(* Logix 5000 project; controller _2081 vendor 1 type 14 code 77 rev 19.11; software revision 19.01 *)

TASK Continuous (continuous, watchdog 500 ms) : BGK_OVEN

MODULES
   Controller : vendor 1 type 14 code 77 (CompactLogixL32EController 0, rev 19.11)
      LocalENB : 1769-L32E Ethernet Port (CompactLogixL32Ethernet 1, rev 19.11)
      Local : CompactBus (CompactVirtualAdapter 3, rev 19.11)
         DC_Input_Slot_3 : 1769-IQ16 (Compact 3, rev 1.1, Input RPI 2 ms)
         DC_Input_Slot_4 : 1769-IQ16 (Compact 4, rev 1.1, Input RPI 2 ms)
         Relay_Out_Slot_5 : 1769-OW8I (Compact 5, rev 2.1, Output RPI 2 ms)
         Analog_Input : 1769-IF8 (Compact 1, rev 1.1, Output RPI 2 ms)
         Analog_Out : vendor 1 type 10 code 39 (Compact 2, rev 1.3, Output RPI 2 ms)
         Relay_Out_Slot_6 : 1769-OW8I (Compact 6, rev 2.1, Output RPI 2 ms)
END_MODULES

TYPE Conveyor :
STRUCT
   Conveyors_Input : PowerFlex_40_Status;
   Conveyor_Output : PowerFlex_40_Command;
END_STRUCT
END_TYPE

TYPE DeviceNETPowerFlex40 :
STRUCT
   Command : PowerFlex_40_Command;   // Start/Stop/Speed Etc.
   Status : PowerFlex_40_Status;   // Fault/Inputs Etc.
END_STRUCT
END_TYPE

TYPE PowerFlex_40_Command :
STRUCT
   Stop : BOOL;   // Stop=1
   Start : BOOL;   // Start=1
   Jog : BOOL;   // Jog=1
   Clear_Faults : BOOL;
   Direction_Forward : BOOL;
   Direction_Reverse : BOOL;
   Not_Used : BOOL;
   MOP_Increment : BOOL;
   Accel_Rate1 : BOOL;
   Accel_Rate2 : BOOL;
   Decel_Rate1 : BOOL;
   Decel_Rate2 : BOOL;
   Reference_Sel1 : BOOL;
   Reference_Sel2 : BOOL;
   Reference_Sel3 : BOOL;
   MOP_Decrement : BOOL;
   Speed_Command : INT;
END_STRUCT
END_TYPE

TYPE PowerFlex_40_Status :
STRUCT
   Ready : BOOL;   // Ready=1
   Active : BOOL;   // Active=1
   Command_Direction : BOOL;   // Forward=1
   Actual_Direction : BOOL;
   Accelerating : BOOL;
   Decelerating : BOOL;
   Alarm_Present : BOOL;
   Fault_Present : BOOL;
   At_Speed : BOOL;
   Main_Freq : BOOL;   // Comm Control=1
   Operation_Command : BOOL;   // Comm Control=1
   Parameters : BOOL;   // Locked=1
   Dig_In_1_Status : BOOL;   // Status of Input 1
   Dig_In_2_Status : BOOL;   // Status of Input 2
   Dig_In_3_Status : BOOL;   // Status of Input 3
   Dig_In_4_Status : BOOL;   // Status of Input 4
   Conveyor_Speed : INT;
END_STRUCT
END_TYPE

VAR_GLOBAL   (* controller tags *)
   Exhaust_Temp_PID : PID := (CTL := -2147446144, EN := 1, INI := 1, OLH := 1, DVPA := 1, PVHA := 1, SP := 300.0, KP := 15.0, KI := 0.2, MAXS := 932.0, MINS := 32.0, SO := 100.0, MAXO := 100.0, UPD := 0.5, PV := 297.0, ERR := 3.0, OUT := 100.0, MAXI := 932.0, MINI := 32.0, MAXCV := 300.0, MAXTIE := 4095.0, DATA[0] := 94.97618, DATA[1] := -471.1111, DATA[2] := 297.0, DATA[3] := 3.0, DATA[4] := 300.0, DATA[5] := 0.11111111, DATA[6] := 1.0, DATA[7] := 8.0, DATA[8] := 15.0, DATA[9] := 0.2, DATA[11] := 15.0, DATA[12] := 0.2, DATA[15] := 3.0, DATA[16] := 0.024420025);
   Exhaust_Temp_PID_Pwr_OUT : DINT := 300;   // PID % Power Out (0-100%)
   Exhaust_Temp_PV : DINT := 297;
   N29 : DINT[4] := ([0] := 1, [1] := 5);
END_VAR

PROGRAM BGK_OVEN   (* main routine mcpMain *)
VAR
   B10 : DINT[255];   // Product Shift Register
   B23 : DINT[20];   // Fault Bits
        [1].13   // Oven Lift Disconnect Fault
        [3].7   // Part On Spindle Before Loader Fault
        [1].17   // MCR NOT ON FAULT
        [4].11   // Booth #2 Low Powder
        [1].1   // P2 Low Temp Warning
        [0].30   // T2 IR Exhaust Air-Flow Fault
        [0]   // Fault Bits Word 0
        [1].10   // Oven Zone6 LampOut Fault
        [4].13   // Unloader Line-Stop Fault
        [3].6   // Conveyor Jam/Take-Up Fault
        [0].13   // Exhaust VFD Fault
        [0].26   // T2 IR Supply #1 MS Fault
        [5].10   // System Shorted SCR Fault
        [4].14   // Spray Booth Line-Stop Fault
        [0].27   // T2 IR Supply #1 Air-Flow Fault
        [1].6   // P2 High Temp Warning
        [5].11   // Zone 2 Shorted SCR Fault
        [5].12   // Zone 3 Shorted SCR Fault
        [0].1   // PLC Battery Low
        [0].29   // IR Exhaust VFD Fault
        [5].1   // CUSTOM: Power Brush VFD Fault
        [0].28   // T2 IR Supply #1 Air-Flow Switch Fault
        [5].13   // Zone 4 Shorted SCR Fault
        [4].6   // Booth #1 Fire
        [1].7   // P3 High Temp Warning
        [0].2   // IR Supply MS Fault
        [4].7   // Booth #1 Not Ready
        [3].10   // Spindle NOT Seated at Loader Fualt
        [1].12   // Remote Console E-Stop
        [4].8   // Booth #1 Low Powder
        [4].10   // Booth #2 Not Ready
        [3].11   // Filter Jammed at Loader Screw Fault
        [1].8   // P4 High Temp Warning
        [5].14   // Zone 5 Shorted SCR Fault
        [1].14   // Oven Lift Open Fault
        [3].1   // IR Conveyor VFD Disconnect Fault
        [1].9   // P5 High Temp Warning
        [5].15   // Zone 6 Shorted SCR Fault
        [4].12   // Loader Line-Stop
        [4].15   // Oven Doors Open Fault
        [3].9   // Bearing Missing Fault
        [2].10   // EXIT PART STOPPED FAULT
        [4].0   // E-Stop Pressed Fault
        [2].7   // Oven Conveyor VFD Faulted
        [4].9   // Booth #2 Fire Detect
        [1].18   // T2 IR Supply #2 Air-Flow Switch Fault
        [5].0   // E-Stop Pressed Fault
        [1]   // B23[xx] ContainsSystem Fault Bits
        [2].9   // ENTRANCE PART STOPPED FAULT
        [3].3   // Exhaust VFD Disconnect Fault
        [1].0   // P1 Low Temp Warning
        [0].15   // Entrance Exhaust Air-Flow Switch Fault
        [0].14   // Exhaust Air-Flow Fault
        [6].4   // Seam Heater Actuator No-Movement Fault
        [3].8   // Part Holder to High Before Loader
        [2].8   // Cooldown Conveyor VFD Faulted
        [3].19   // T2 Exhaust VFD Disconnect Fault
        [0].11   // Recirculation Air-Flow Fault
        [3].13   // Oven Conveyor Motion Fault
        [1].5   // P1 High Temp Warning
        [3].4   // PEG Conveyor VFD Disconnect Fault
        [1].2   // P3 Low Temp Warning
        [1].11   // Main CB UV Trip Disabled Fault
        [3].12   // IR Conveyor Motion Fault
        [3].15   // Seam Heater Crash Detect Fault
        [0].12   // Recirculation Air-Flow Switch Fault
        [3].14   // Cooldown Conveyor Motion Fault
        [3].2   // Cooldown Conveyor VFD Disconnect Fault
        [1].16   // OVEN CONVEYOR NOT ON FAULT
        [1].24   // Control Panel Door E-Stop Fault
        [1].15   // MAIN CAB DISC OFF OR HIGH TEMP LIMIT IS TRIPPED FAULT
        [3].5   // T2 Exhaust VFD Disconnect Fault
        [1].3   // P4 Low Temp Warning
        [1].4   // P5 Low Temp Warning
        [0].5   // Temperature Deviation Fault
        [0].6   // Oven Overtemp Limit Fault
        [0].7   // Hot-Air Contactor #1 Fault
        [0].8   // Hot-Air Contactor #2 Fault
        [0].10   // Recirculation VFD Fault
   B3 : DINT[10] := ([0] := 2#0000_0000_0000_0000_0000_1000_0000_1010, [1] := 2#0000_0000_0000_0000_0000_0001_0000_0110, [3] := 2#0000_0000_0000_0000_0000_0000_0100_0001);   // Utility Bits
        [1].10   // Idle Force ON One-Shot
        [0].11   // Oven is in Cooldown Mode
        [1].5   // Oven Motion Low Pulse
        [0].10   // USE PID or OLD Code ( 1 == OLD Code)
        [0].6   // Spare
        [1].4   // Oven Motion HIGH Pulse
        [0].3   // NO Air-Flow Faults
        [0].4   // Spare
        [0].25   // Enable OK to Take Temperature Audible
        [0].12   // Spare
        [0].2   // Spare
        [0].8   // Spare
        [0].0   // Motion Shift One-Shot
        [0].1   // Conveyor Motion Simulate
        [0].13   // Maintain Conveyor RUN One-Shot
        [0].15   // System Auto-Stop One-Shot
        [1].11   // Idle Force OFF One-Shot
        [1].0   // Closed-Loop Enable IR Section #1
        [0].5   // Oven Blowers are ON
        [1].1   // Closed-Loop Enable IR Section #2
        [1].2   // Closed-Loop Enable IR Section #3
        [0].7   // O.K. to Take Part Peak Temperature
        [0].16   // Spare
        [0].17   // Spare
        [0].9   // Part Passing Through FIFO One-Shot
        [1].8   // Use OLD (BGK Developed) PID
        [0].14   // System was Auto-Started Last Scan
        [0].24   // 14s Audible Enable
        [0].19   // Horn Silence/Reset Secondary Condition
        [0].20   // Horn Silence/Reset Secondary Condition
        [0].18   // Horn Silence/Reset Secondary Condition
   B33 : DINT[10] := ([0] := 2#0000_0000_0000_0000_0100_1100_0000_1100, [1] := 2#1111_1111_1111_1111_0000_0001_0000_1001, [2] := 2#0000_0000_0000_0000_0000_0000_0000_0111, [6] := 2#0000_0000_0000_0000_0000_0000_0000_0100);   // Utility Bits
        [6].6   // Oven Purging
        [6].9   // System Ready
        [1].14   // Alarm Horn Compare
        [0].4   // Conveyor Motion
        [6].3   // System in Manual
        [0].7   // Silence/ Reset One-Shot
        [0].2   // UV Enable
        [1].9   // Part Holder Detected Latch
        [0].10   // NO Oven Conveyor Faults
        [0].8   // Oven Purge Done
        [0].12   // Any Air-Flow Fault
        [2].1   // Alarm Horn Compare Result
        [0].11   // NO Cooldown Conveyor Faults
        [2].2   // Alarm Light Compare Result
        [0].13   // Any Exhaust Fault
        [6].1   // Main Power Off
        [6].2   // MCR Power Off
        [6].8   // Oven in Cooldown
        [6].4   // System in Auto
        [2].0   // Alarm Control
        [0].3   // MCR Enable
        [0].15   // ANY OVEN Fault
        [0].0   // ALWAYS FALSE TEST BIT
        [1].11   // IR Oven Manual Idle Control
        [0].29   // Any Exhaust Fault
        [1].4   // Any Power Brush Fault
        [6].5   // Auto-Start
        [6].10   // System Running
        [0].5   // Booth #1 Selected
        [0].16   // IR Conveyor Running
        [1].7   // Recipe Between 26 & 50
        [0].6   // Booth #2 Selected
        [1].2   // Seam Heater Auto OUT
        [1].8   // Spindle Detected Latch
        [0].18   // Any Conveyor Line-Stop Fault
        [6].7   // Purging Done - Start Conveyor
        [0].14   // T2 Any IR Conveyor Fault
        [1].1   // Seam Heater Auto IN
        [1].15   // Alarm Light Control
        [2].4   // Alarm Reset Pulse
        [1].0   // Seam Heater Auto Position Move Complete
        [0].1   // IR Entrance Part Detected
        [0].9   // Oven Was ON Last Scan
        [0].20   // IR Conveyor Line Re-Start One-Shot
        [1].3   // No Product In Zones 1,2 or 3
        [1].10   // IR Oven Manual Run Control
   B36 : DINT[10] := ([0] := 2#0000_0000_1000_0000_0000_0000_0000_0000, [1] := 2#0000_0000_0000_0000_0000_1000_0000_0000, [2] := 2#0000_0000_0000_0000_0000_0000_0001_0010);   // One-Shots
        [0].22   // One-Shot
        [0].23   // One-Shot
        [1].9   // One-Shot
        [0].17   // One-Shot
        [0].10   // One-Shot
        [0].6   // Used One-Shot
        [0].7   // Used One-Shot
        [0].0   // One-Shot
        [0].1   // One-Shot
        [0].2   // One-Shot
        [0].3   // One-Shot
        [0].4   // One-Shot
        [0].5   // One-Shot
        [0].11   // One-Shot
        [0].9   // One-Shot
        [0].15   // oneshot
        [0].12   // One-Shot
        [1].0   // One-Shot
        [0].13   // One-Shot
        [1].1   // One-Shot
        [1].2   // One-Shot
        [0].14   // One-Shot
        [1].3   // One-Shot
        [2].0   // One-Shot
        [0].18   // One-Shot
        [2].1   // One-Shot
        [1].10   // One-Shot
        [2].2   // One-Shot
        [1].11   // One-Shot
        [2].3   // One-Shot
        [2].4   // One-Shot
        [1].12   // One-Shot
        [0].8   // Used One-Shot
        [1].17   // One-Shot
        [2].5   // One-Shot
        [1].5   // One-Shot
        [1].6   // One-Shot
        [1].4   // One-Shot
        [1].16   // One-Shot
        [1].13   // One-Shot
        [1].14   // One-Shot
        [1].15   // One-Shot
        [0].16   // One-Shot
   B37 : DINT[10];   // Product Location
        [0].13   // IR Section 10 Product Present
        [0].4   // IR Section 1 Product Present
        [0].5   // IR Section 2 Product Present
        [0].1   // Product Present Gun #1
        [0].2   // Product Present Gun #2
        [0].14   // IR Section 11 Product Present
        [0].3   // Product Present Gun #3
        [0].15   // IR Section 12 Product Present
        [0].6   // IR Section 3 Product Present
        [0].8   // IR Section 5 Product Present
        [0].9   // IR Section 6 Product Present
        [0].10   // Cooldown Section Product Present
        [0].0   // Powder Booth Part Present
        [1].5   // Booth 2 Gun 1 OK to Spray
        [0].11   // IR Section 8 Product Present
        [1].6   // Booth 2 Gun 2 OK to Spray
        [0].7   // Cooldown Product Present
        [0].12   // IR Section 9 Product Present
   C35 : COUNTER[5] := ([0].PRE := 6, [3].PRE := 30, [4].PRE := 8);   // Closed-Loop Counters
        [0]   // Closed-Loop #1 FIFO Counter
        [1]   // Closed-Loop #2 FIFO Counter
        [3]   // Peak-Picker Delay Counter
        [4]   // Peak-Picker Duration Counter
        [0].PRE   // Closed-Loop#1 FIFO Counter
   C5 : COUNTER[15] := ([0].PRE := 80, [0].ACC := 3431, [1].PRE := 3, [1].ACC := 3419, [2].PRE := 3, [2].ACC := 3416, [3].PRE := 3, [3].ACC := 3416, [4].PRE := 180, [4].ACC := 140187, [4].DN := 1, [5].PRE := 180, [5].ACC := 140138, [5].DN := 1, [6].PRE := 180, [6].ACC := 140068, [6].DN := 1, [7].PRE := 200, [7].ACC := 3341, [8].PRE := 2, [9].PRE := 4000, [9].ACC := 4147, [9].DN := 1, [10].PRE := 2000, [10].ACC := 4138, [10].DN := 1, [11].PRE := 6, [11].ACC := 7, [12].PRE := 6, [12].ACC := 3);   // Line Duration Counters
        [1]   // Spare
        [0]   // Spare
        [4]   // IR Section 1 Duration
        [5]   // IR Section 2 Duration
        [6]   // IR Section 3 Duration
        [10]   // Cooldown Blower Duration
        [2]   // Spare
        [2].PRE   // Gun 2 Duration
        [3]   // Spare
        [8]   // Spare
        [7]   // Spare
        [12]   // Spare
        [11]   // Spare
        [13]   // Spare
        [14]   // Spare
        [9]   // FIFO Reset Counter
   CLDN_Conveyor_Speed_Reference : INT := 26115;   // DIGITAL COMMAND TO COOLDOWN CONVEYOR VFD
   DeviceNET_Scanner_Enable : BOOL := 1;
   Exhaust_Speed_Reference : INT := 31500;   // EXHAUST VFD Digital Command Speed
   F38 : REAL[25] := ([1] := 3.0, [11] := 0.5, [15] := 4.0);
        [1]   // Closed-Loop #1 Proportional Multiplier
        [0]   // Closed-Loop #1 Accumulator
        [3]   // Closed-Loop #2 Proportional Multiplier
        [2]   // Closed-Loop #2 Accumulator
        [17]   // Conveyor Speed Actual Display
        [15]   // Conveyor Speed Set Display
        [16]   // Cooldown Speed Set Display
        [11]   // Closed-Loop Integral Accumulator
        [18]   // Cooldown Speed Actual Display
   F8 : REAL[5] := ([0] := 8.038388, [1] := 17227.26);   // Floating Point (Real)
        [0]   // Oven ON Time in Hours
        [1]   // Oven OFF Time in Minutes
   i1 : INT[8] := ([0] := 678, [1] := 715, [2] := 720, [3] := 734, [4] := 761, [5] := 2954, [6] := 1, [7] := 2);   // 8-pt Analog Inputs
        [7]   // Spare 0-10Vdc Input
        [1]   // Oven Exit Pyrometer #2 (0-5Vdc; 32-932f)
        [6]   // Customer Conveyor Speed Reference (0-10Vdc)
        [2]   // Oven Exit Pyrometer #3 (0-5Vdc; 32-932f)
        [3]   // Oven Exit Pyrometer #4 (0-5Vdc; 32-932f)
        [4]   // Oven Exit Pyrometer #5 (0-5Vdc; 32-932f)
        [5]   // Hot-Air Oven Process Temperature Feedback (0-10Vdc; 32-932f)
        [0]   // Oven Exit Pyrometer #1 (0-5Vdc; 32-932f)
   i3 : INT := 11295;   // Slot 3 16pt DC Input
        .9   // Oven Exit Product Detect
        .0   // MCR Status
        .5   // Oven Exhaust Blower Differential Air-Flow SW
        .6   // Spare
        .2   // Oven Lift MS Aux. Input
        .7   // Oven Recirculation Blower Differential Air-Flow SW
        .3   // Infeed Conveyor Running
        .1   // Main CB Status
        .8   // Oven Entrance Product Detect
        .10   // Oven Conveyor VFD Status
        .12   // Spare
        .13   // Oven Recirculation VFD Status
        .11   // Oven Exhaust VFD Status
        .4   // Outfeed (Exit) Conveyor Running
        .14   // Oven Overtemp Limit (1==FAULT)
        .15   // Oven Temperature Deviation Warning
   i4 : INT := 16;   // Slot 4 16pt DC Input
        .1   // Spare
        .2   // Spare
        .13   // Spare
        .14   // Spare
        .3   // Spare
        .10   // Spare
        .15   // Spare
        .4   // Conveyor Motion Proximity Sensor
        .5   // Duct Heater Contactor #1Aux. Input
        .12   // Spare
        .7   // Spare
        .6   // Duct Heater Contactor #2Aux. Input
        .9   // Spare
        .8   // Spare
        .11   // Spare
        .0   // Spare
   IR_1_BITOff : DINT := 5;   // Indirect Addressing BIT Offset
   IR_1_DWOff : DINT := 4;   // Indirect Addressing WORD Offset
   IR_BITOff : DINT := 24;
   IR_Conveyor_Speed_Reference : INT := 26850;   // DIGITAL COMMAND TO OVEN CONVEYOR VFD
   IR_DWOff : DINT := 3;
   N18 : DINT[205] := ([25] := 246, [26] := 240, [27] := 238, [28] := 240, [29] := 233, [30] := 231, [31] := 228, [32] := 228, [33] := 230, [34] := 227, [35] := 243, [36] := 242, [37] := 236, [38] := 241, [39] := 240, [40] := 242, [41] := 235, [42] := 241, [43] := 234, [44] := 234, [45] := 233, [46] := 237, [47] := 238, [48] := 241, [49] := 243, [50] := 236, [51] := 246, [52] := 232, [53] := 238, [54] := 242, [55] := 232, [56] := 228, [57] := 227, [58] := 238, [59] := 236, [60] := 229, [61] := 242, [62] := 243, [63] := 240, [64] := 236, [65] := 241, [66] := 232, [67] := 231, [68] := 234, [69] := 234, [70] := 236, [71] := 231, [72] := 235, [73] := 231, [74] := 226, [75] := 228, [76] := 228, [77] := 234, [78] := 228, [79] := 233, [80] := 234, [81] := 238, [82] := 238, [83] := 245, [84] := 239,
        [85] := 232, [86] := 239, [87] := 234, [88] := 230, [89] := 232, [90] := 225, [91] := 225, [92] := 224, [93] := 231, [94] := 226, [95] := 229, [96] := 237, [97] := 240, [98] := 233, [99] := 227, [100] := 237, [101] := 245, [102] := 248, [103] := 244, [104] := 235, [105] := 232, [106] := 231, [107] := 229, [108] := 233, [109] := 232, [110] := 234, [111] := 247, [112] := 239, [113] := 236, [114] := 238, [115] := 230, [116] := 229, [117] := 226, [118] := 229, [119] := 236, [120] := 242, [121] := 238, [122] := 251, [123] := 240, [124] := 246, [125] := 240, [126] := 238, [127] := 240, [128] := 233, [129] := 231, [130] := 228, [131] := 228, [132] := 230, [133] := 227, [134] := 243, [135] := 242, [136] := 236, [137] := 241, [138] := 240, [139] := 242, [140] := 235, [141] := 241, [142] := 234, [143] := 234, [144] := 233,
        [145] := 237, [146] := 238, [147] := 241, [148] := 243, [149] := 236, [150] := 246, [151] := 232, [152] := 238, [153] := 242, [154] := 232, [155] := 228, [156] := 227, [157] := 238, [158] := 236, [159] := 229, [160] := 242, [161] := 243, [162] := 240, [163] := 236, [164] := 241, [165] := 232, [166] := 231, [167] := 234, [168] := 234, [169] := 236, [170] := 231, [171] := 235, [172] := 231, [173] := 226, [174] := 228, [175] := 228, [176] := 234, [177] := 228, [178] := 233, [179] := 234, [180] := 238, [181] := 238, [182] := 245, [183] := 239, [184] := 232, [185] := 239, [186] := 234, [187] := 230, [188] := 232, [189] := 225, [190] := 225, [191] := 224, [192] := 231, [193] := 226, [194] := 229, [195] := 237, [196] := 240, [197] := 233, [198] := 227, [199] := 225);   // Closed-Loop #1 FIFO
        [100]   // Closed-Loop #1 FIFO Temporary Shift Area
        [0]   // Closed-Loop #1 FIFO
        [1]   // Closed-Loop #1 FIFO
   N19 : DINT[205] := ([0] := 244, [1] := 237, [2] := 245, [3] := 248, [4] := 244, [5] := 235, [6] := 232, [7] := 231, [8] := 229, [9] := 233, [10] := 232, [11] := 234, [12] := 247, [13] := 239, [14] := 236, [15] := 238, [16] := 230, [17] := 229, [18] := 226, [19] := 229, [20] := 236, [21] := 242, [22] := 238, [23] := 251, [24] := 240, [25] := 246, [26] := 240, [27] := 238, [28] := 240, [29] := 233, [30] := 231, [31] := 228, [32] := 228, [33] := 230, [34] := 227, [35] := 243, [36] := 242, [37] := 236, [38] := 241, [39] := 240, [40] := 242, [41] := 235, [42] := 241, [43] := 234, [44] := 234, [45] := 233, [46] := 237, [47] := 238, [48] := 241, [49] := 243, [50] := 236, [51] := 246, [52] := 232, [53] := 238, [54] := 242, [55] := 232, [56] := 228, [57] := 227, [58] := 238, [59] := 236,
        [60] := 229, [61] := 242, [62] := 243, [63] := 240, [64] := 236, [65] := 241, [66] := 232, [67] := 231, [68] := 234, [69] := 234, [70] := 236, [71] := 231, [72] := 235, [73] := 231, [74] := 226, [75] := 228, [76] := 228, [77] := 234, [78] := 228, [79] := 233, [80] := 234, [81] := 238, [82] := 238, [83] := 245, [84] := 239, [85] := 232, [86] := 239, [87] := 234, [88] := 230, [89] := 232, [90] := 225, [91] := 225, [92] := 224, [93] := 231, [94] := 226, [95] := 229, [96] := 237, [97] := 240, [98] := 233, [99] := 227);   // Previous Closed-Loop Part Temperature Values
        [100]   // Closed-Loop #2 Pyrometer Peak-Picker
        [0]   // Previous Closed-Loop Part Temperature Values
   N21 : DINT[50] := ([0] := 480, [1] := 340, [3] := 100, [4] := 550, [5] := 100, [6] := 100, [7] := 150, [10] := 50, [12] := 32767, [13] := 6241, [14] := 31206, [16] := 600, [17] := 15, [20] := 784, [21] := 784, [22] := 466, [23] := 5, [24] := 3, [30] := 65535, [31] := -65536, [32] := 120, [33] := 6144, [35] := 75, [36] := 150, [37] := 300, [40] := 10);   // Configuration Values
        [2]   // Recipe Edit Minimum Voltage
        [22]   // Shift Register Password
        [1]   // System Maximum Line Speed
        [4]   // Maximum Set Exit Temperature
        [3]   // Maximum Rotator Speed
        [15]   // 0-10v Analog-In Scaled Minimum Value
        [6]   // Duct Heater % Power
        [13]   // 0-10v Analog-In Minimum Value
        [7]   // Cooldown Temperature Setpoint
        [11]   // 0-10v Analog-Out Minimum Value
        [24]   // Minimum Scaled Seam Mover Movement Required to Prevent Fault
        [14]   // 0-10v Analog-In Maximum Value
        [20]   // Recipe Edit Password
        [12]   // 0-10v Analog-Out Maximum Value
        [23]   // Seam Heater Dead-Band
        [33]   // E-Stop (MCR) Fault Compare Mask
        [5]   // Maximum Power-Brush Speed
        [32]   // Closed-Loop Peak-Picker Minimum Value
        [21]   // System Setup Password
        [10]   // Recipe Length
        [0]   // System Max. Voltage -380,415,480,575
        [42]   // Shift Register Password
        [31]   // High 2-Byte Mask
        [41]   // Maximum Deviation Allowed for Lamp-Out
        [30]   // Low 2-Byte Mask
        [40]   // Maximum Deviation Allowed to Shorted SCR ma x 10
        [16]   // 0-10v Analog-In Scaled Maximum Value
        [36]   // Lower Bound for Temperature Window
        [37]   // Upper bound for Temperature Window
        [35]   // Temperature Window Size
        [17]   // Exhaust VFD Integral Enable Temperature Window
   N26 : DINT[600] := ([0] := 88, [5] := 1024, [21] := 784, [24] := 10, [25] := 140, [26] := 66, [27] := 300, [28] := 1, [29] := 10, [30] := 20, [31] := 1, [32] := 45, [33] := 1, [35] := 30, [37] := 100, [38] := 21, [39] := 420, [40] := 150, [41] := 50, [42] := 10, [43] := 75, [44] := 40, [50] := 67, [51] := 100, [52] := 45, [53] := 75, [54] := 200, [60] := 200, [61] := 200, [62] := 200, [63] := 200, [64] := 200, [65] := 200, [68] := 100, [71] := 500, [72] := 500, [73] := 500, [74] := 500, [75] := 500, [76] := 115, [77] := 75, [78] := 125, [79] := 101, [81] := 100, [82] := 100, [83] := 100, [84] := 100, [85] := 100, [100] := 80, [101] := 180, [102] := 180, [103] := 180, [104] := 180, [105] := 70, [106] := 20, [107] := 200, [108] := 20, [109] := 20, [110] := 2000, [120] := 10,
        [121] := 22, [122] := 25, [123] := 28, [124] := 1, [125] := 50, [126] := 120, [127] := 100, [128] := 60, [129] := 70, [132] := 65, [133] := 24, [145] := 133, [180] := 500, [181] := 500, [200] := 6, [201] := 75, [202] := 30, [204] := 15000, [208] := 175, [212] := 10, [300] := 330, [301] := 330, [303] := 330, [304] := 330, [340] := 40, [341] := 120, [342] := 45, [343] := 75, [345] := 5, [346] := 8, [500] := 1, [501] := 5, [502] := 1, [503] := -1, [510] := 1, [512] := 50, [513] := 35, [514] := 3, [515] := -35);   // Write to PLC
        [1].0   // Auto Start Ststem (Momentary PB)
        [0].6   // Line-Start Boost Enabled
        [24]   // Remote Recipe Select From Customer's PLC (1-50)
        [4].11   // Part Feed Stop PB
        [0].5   // IR Oven Manual Idle PB
        [510]   // Exhaust VFD Integral Correction (Up or Down)
        [513]   // Exhaust VFD Maximum Closed-Loop Total Sum
        [0].2   // Horn Silence/ Fault Reset
        [1].1   // Recirculation Manual Start
        [1].9   // Accumulator Conveyor Start PB
        [1].17   // T2 IR Supply #1 Manual Start
        [1].19   // T2 IR Supply #2 Manual Start
        [4].7   // B1 Powder Robber Manual Stop
        [4].8   // B2 Powder Robber Manual Stop
        [5].1   // IR Idle Force
        [60]   // Manual IR Voltages
        [0].3   // Duct Heater Enable == 0 Disable == 1
        [0].4   // Filter Down Fault Bypass
        [3].1   // Oven Conveyor Manual Start
        [3].11   // Part Feed Start PB
        [1].13   // MagDown Conveyor Start PB
        [1].6   // Duct Heater Manual Start
        [50]   // Manual Oven Conveyor Speed
        [2].2   // Exhaust VFD Manual Stop
        [1].5   // Oven Manual Run PB
        [2].5   // Oven Manual Stop PB
        [103]   // IR Section 3 Duration
        [1].7   // Loader Infeed Start PB
        [2].6   // Duct Heater Manual Stop
        [1].2   // Exhaust VFD Manual Start
        [1].10   // MagUp Conveyor Start PB
        [61]   // Manual IR Voltages
        [2].9   // Accumulator Conveyor Stop PB
        [10]   // BIT USE
        [3].7   // B1 Powder Robber Manual Start
        [2].11   // Mez Feed Conveyor Stop PB
        [0]   // BIT USE
        [2].17   // T2 IR Supply #1 Manual Stop
        [0].0   // System in Auto/Manual (0 == Auto)
        [0].7   // LampOut Fault Bypass
        [3].3   // T2 Conveyor Manual Start
        [62]   // Manual IR Voltages
        [11]   // BIT USE
        [2].12   // Mez Exit Conveyor Stop PB
        [1]   // BIT USE
        [0].1   // System Auto-Start Momentary P.B.
        [204]   // C.L. #1 Maximum Line-Stopped Time Before Resetting FIFO Counter
        [3].4   // Manual Start B1 Gun 2
        [63]   // Manual IR Voltages
        [12]   // BIT USE
        [2]   // BIT USE
        [1].11   // Mez Feed Conveyor Start PB
        [214]   // C.L. #2 Maximum Line-Stopped Time Before Resetting FIFO Counter
        [2].8   // Infeed Metering Conveyor Stop PB
        [4].9   // B1 Blow-Off Manual Stop
        [3].5   // Manual Start B1 Gun 3
        [64]   // Manual IR Voltages
        [20]   // Recipe Edit Password
        [22]   // Shift Register Password
        [13]   // BIT USE
        [3]   // BIT USE
        [42]   // Line-Start Boost Time Constant (tau)
        [4].17   // T2 Conveyor Manual Stop
        [65]   // Manual IR Voltages
        [2].13   // MagDown Conveyor Stop PB
        [14]   // BIT USE
        [4]   // BIT USE
        [5].4   // Shift Register Edit Data Notify
        [0].8   // Reset Seam Heater Raw Max. Value
        [41]   // Boost Power Max. Percent %
        [101]   // IR Section 1 Duration
        [66]   // Manual IR Voltages
        [202]   // Closed-Loop Proportional Multiplier
        [4].0   // Conveyors Auto-Stop
        [33]   // Recipe-to-Run From PV
        [2].19   // T2 IR Supply #2 Manual Stop
        [5].5   // Accept New Recipe Value From CTC
        [2].10   // MagUp Conveyor Stop PB
        [1].8   // Infeed Metering Conveyor Start PB
        [102]   // IR Section 2 Duration
        [67]   // Manual IR Voltages
        [124]   // IR Section 1 Start Point
        [4].12   // B1 Air-Knife Manual Stop
        [3].9   // B1 Blow-Off Manual Start
        [4].3   // T2 Conveyor Manual Stop
        [3].6   // Manual Start B2 Gun 2
        [68]   // Manual IR Voltages
        [40]   // IR Idle Voltage
        [2].7   // Loader Infeed Stop PB
        [35]   // Screen Status From PV
        [125]   // IR Section 2 Start Point
        [121]   // B1 Gun 1 Start Position
        [69]   // Manual IR Voltages
        [4].13   // B2 Air-Knife Manual Stop
        [31]   // Recipe Edit Pointer
        [126]   // IR Section 3 Start Point
        [201]   // Maximum CL #1 Voltage Correction
        [122]   // B1 Gun 2 Start Position
        [4].6   // Manual Start B2 Gun 2
        [203]   // Closed-Loop Temperature Setpoint
        [127]   // IR Section 4 Start Point
        [211]   // Maximum CL #2 Voltage Correction
        [4].4   // Manual Stop B1 Gun 2
        [145]   // Closed-Loop #1 Pyrometer Position
        [4].5   // Manual Stop B1 Gun 3
        [128]   // IR Section 5 Start Point
        [146]   // Closed-Loop #2 Pyrometer Position
        [15]   // BIT USE
        [5]   // BIT USE
        [100]   // Powder Booth Duration
        [200]   // Closed-Loop FIFO Length
        [37]   // Manual IR Edit Value
        [1].12   // Mez Exit Conveyor Start PB
        [5].3   // IR Manual Edit Data Notify
        [16]   // BIT USE
        [6]   // BIT USE
        [5].11   // Clear Closed-Loop #1 FIFO
        [1].18   // T2 IR Exhaust Manual Start
        [21]   // System Setup Password
        [17]   // BIT USE
        [7]   // BIT USE
        [3].8   // B2 Powder Robber Manual Start
        [4].10   // Accum & Unload Conv Auto Stop
        [5].13   // Clear Closed-Loop #2 FIFO
        [210]   // Closed-Loop #2 FIFO Length
        [3].17   // T2 Conveyor Manual Start
        [18]   // BIT USE
        [8]   // BIT USE
        [129]   // IR Section 6 Start Point
        [3].12   // B1 Air-Knife Manual Start
        [5].12   // Closed-Loop #2 Control ON/OFF
        [32]   // Recipe Edit Entered Value
        [19]   // BIT USE
        [9]   // BIT USE
        [3].13   // B2 Air-Knife Manual Start
        [38]   // Shift Register List Pointer
        [212]   // VFD Proportional Multipplier x 10
        [130]   // IR Section 7 Start Point
        [5].10   // Closed-Loop Control ON/OFF
        [131]   // IR Section 8 Start Point
        [5].0   // Recipe Edit Accept One-Shot
        [132]   // IR Section 9 Start Point
        [512]   // Exhaust VFD Maximum Closed-Loop Integral / Proportional Sum
        [133]   // IR Section 10 Start Point
        [502]   // Maximum Closed-Loop Integral Sum
        [34]   // Recipe Edit parameter Select
        [5].2   // Recipe-to-Run Notify From PV
        [501]   // Integral Multiplier (x 10)
        [36]   // Maximum CL Voltage Correction
        [208]   // FIFO C.L. Temperature Setpoint
        [2].0   // Auto Stop System (Momentary PB)
        [2].1   // Recirculation Manual Stop
        [3].2   // Cooldown Conveyor Manual Start
        [3].10   // Accum & Unload Conv Auto Start
        [6].1   // Reset Minute Timer PB
        [1].3   // Exit Exhaust Manual Start
        [2].3   // Exit Exhaust Manual Stop
        [110]   // Cooldown Duration
        [44]   // Exhaust VFD Minimum Auto Speed %
        [2].4   // HEPS Supply Blowers Manual STOP
        [0].10   // Recipe Copy PB
        [0].11   // Local/Remote Recipe Select (0==Local)
        [1].4   // HEPA Supply Blowers Manual Start
        [28]   // Recipe Copy
        [0].9   // Local/Remote Line Speed Command (0==Local)
        [29]   // Recipe Copy
        [3].0   // Conveyor Auto Start
        [4].2   // Cooldown Conveyor Manual Stop
        [30]   // Recipe To Edit Display Pointer
        [500]   // Integral Correction (Up or Down)
        [52]   // Exhaust VFD Manual Speed
        [6].0   // Reset Hour Timer PB
        [39]   // Oven Warm-Up Voltage
        [503]   // Minimum Closed-Loop Integral Sum
        [23]   // Remote Line-Speed From Customer's PLC (0-340 == 0.0-34.0fpm)
        [4].1   // Oven Conveyor Manual Stop
        [51]   // Manual Oven Temperature Setpoint
        [53]   // Recirculation VFD Manual Speed
        [25]   // Oven Cooldown Temperature Setpoint
        [72]   // Exit Pyrometer #2 High Temp Warning
        [71]   // Exit Pyrometer #1 High Temp Warning
        [73]   // Exit Pyrometer #3 High Temp Warning
        [74]   // Exit Pyrometer #4 High Temp Warning
        [75]   // Exit Pyrometer #5 High Temp Warning
        [26]   // Oven CoolDown Exhaust Speed (0-100%)
        [81]   // Exit Pyrometer #1 Low Temp Warning
        [82]   // Exit Pyrometer #2 Low Temp Warning
        [83]   // Exit Pyrometer #3 Low Temp Warning
        [84]   // Exit Pyrometer #4 Low Temp Warning
        [85]   // Exit Pyrometer #5 Low Temp Warning
   N27 : DINT[400] := ([1] := 4, [2] := 81, [4] := 64, [5] := 1024, [6] := 10, [33] := 1, [34] := 32768, [36] := 230, [40] := 23, [41] := 50, [42] := 10, [45] := 300, [50] := 117, [51] := 71, [52] := 73, [53] := 74, [54] := 74, [55] := 76, [60] := 200, [61] := 200, [62] := 200, [63] := 200, [64] := 200, [65] := 200, [68] := 100, [79] := 51, [101] := 400, [110] := 150, [150] := 400, [151] := 400, [152] := 400, [153] := 400, [154] := 400, [155] := 400, [156] := 400, [157] := 360, [158] := 360, [190] := 40, [191] := 400, [192] := 40, [193] := 100, [195] := 30, [196] := 8, [197] := 1, [198] := 275, [200] := 6, [201] := 75, [202] := 30, [204] := 15000, [206] := 81, [208] := 175, [212] := 10);   // Read from PLC
        [212]   // VFD Exhaust Proportional Multiplier x 10
        [42]   // Line-Start Boost Time Constant (tau) FB
        [20]   // Purge Time Remaining (s)
        [0].1   // Exhaust VFD ON
        [2].5   // Recirculation Air-Flow Switch
        [150]   // Active Recipe Zone 1 Voltage
        [3].0   // Duct Heater Oven ON
        [3].1   // IR Oven Idle Mode
        [2].15   // T2 Supply #1 Air-Flow Switch
        [0].13   // Oven is Purging
        [2].16   // T2 Supply #2 Air-Flow Switch
        [5].3   // IR Manual Edit Data Handshake
        [0].12   // Oven is in Cooldown
        [0].8   // Cooldown 4 Supply MS ON
        [33]   // Recipe-to-Run To PV
        [1].10   // Booth 2 Gun 2 Trigger
        [1].5   // Booth 1 Ready and Selected
        [1].6   // Booth 2 Ready and Selected
        [0].0   // Recirculation MS ON
        [0].6   // Oven Calibrate Control
        [1].11   // B1 Powder Robber Vibrator ON/OFF
        [0]   // BIT USE
        [0].16   // T2 IR Supply #1 MS ON
        [197].0   // Active Recipe Electric Hot-Air ON/OFF
        [201]   // Maximum CL Voltage Correction FB
        [0].18   // T2 IR Supply #2 MS ON
        [0].14   // Oven Purge Complete
        [1]   // BIT USE
        [2].3   // Oven Exit Part Detect Indicator
        [204]   // C.L. #1 Maximum Line-Stopped Time Before Resetting FIFO Counter FB
        [1].7   // Booth 1 Gun 1 Trigger
        [34].0   // EQU
        [2]   // BIT USE
        [44]   // Total Boost % Power to Add to System
        [71]   // Scaled Temperature Feedback (32-932)
        [1].8   // Booth 1 Gun 2 Trigger
        [3]   // BIT USE
        [202]   // Closed-Loop #1 Proportional Multiplier
        [2].10   // MagUp Conveyor Status
        [1].9   // Booth 1 Gun 3 Trigger
        [4]   // BIT USE
        [205]   // Closed-Loop #1 Voltage Correction
        [3].2   // Hot-Air Duct Heater ON
        [0].17   // T2 IR Exhaust VFD ON
        [206]   // C.L. #1 Pyrometer Temperature Feedback
        [203]   // Closed-Loop Temperature Setpoint FB
        [2].14   // T2 Motion Detect Indicator
        [2].17   // T2 Exhaust #1 Air-Flow Switch
        [119]   // T2 IR Zone 10 Run Value
        [1].0   // System Auto-Started
        [5].2   // Recipe-to-Run Notify To PV
        [120]   // T2 IR Zone 11 Run Value
        [300]   // Closed-Loop Integral Correction
        [121]   // T2 IR Zone 12 Run Value
        [122]   // T2 IR Zone 1 Run Value
        [1].4   // Booth #2 Ready to PV
        [1].13   // B1 Blow-Off ON/OFF
        [35]   // Screen Control To PV
        [159]   // Active Recipe Value 10
        [123]   // T2 IR Zone 2 Run Value
        [1].14   // B2 Blow-Off ON/OFF
        [160]   // Active Recipe Value 11
        [124]   // T2 IR Zone 3 Run Value
        [5].4   // Shift Edit Handshake
        [161]   // Active Recipe Value 12
        [0].7   // Cooldown 3 Exhaust MS ON
        [162]   // Active Recipe Value 13
        [125]   // T2 IR Zone 4 Run Value
        [5]   // BIT USE
        [163]   // Active Recipe Value 14
        [1].12   // B2 Powder Robber Vibrator ON/OFF
        [164]   // Active Recipe Value 15
        [6]   // BIT USE
        [1].17   // T2 Conveyor Run Indicator
        [5].10   // Closed-Loop #1 Control ON/OFF FB
        [6].0   // Main Power Status Ind
        [2].0   // Power Brush VFD RUN
        [7]   // BIT USE
        [2].11   // Mez Feed Conveyor Status
        [2].1   // B1 Air-Knife ON/OFF
        [6].2   // Powder Booth Not Ready Ind
        [8]   // BIT USE
        [5].12   // Closed-Loop #2 Control ON/OFF FB
        [1].3   // T2 Conveyor Run Indicator
        [165]   // Active Recipe Value 16
        [36]   // Hot-Air Temperature Setpoint
        [0].15   // Auto/Manual to PV (0==Auto)
        [207]   // C.L. #1 FIFO Ave. To PV
        [166]   // Active Recipe Value 17
        [9]   // BIT USE
        [126]   // T2 IR Zone 5 Run Value
        [127]   // T2 IR Zone 6 Run Value
        [167]   // Active Recipe Value 18
        [168]   // Active Recipe Value 19
        [3].6   // Line-Start Boost Enabled FB
        [169]   // Active Recipe Value 20
        [4].6   // Line-Start Boost Enabled FB
        [34]   // Recipe Parameter Select to PV
        [302]   // Closed-Loop Integral Sum
        [2].12   // Mez Exit Conveyor Status
        [41]   // Boost Power Max. Percent % FB
        [192]   // Active Recipe - Bit Defined
        [110]   // IR Zone 1 Run Value
        [111]   // IR Zone 2 Run Value
        [2].4   // Oven Conveyor Motion Detect Indicator
        [155]   // Active Recipe Zone 6 Voltage
        [53]   // Oven Exit Pyrometer Temperature #3 Feedback (0-5Vdc == 32-932f)
        [0].4   // HEPA Supply Blower RUN Status
        [54]   // Oven Exit Pyrometer Temperature #4 Feedback (0-5Vdc == 32-932f)
        [0].11   // Recipe Select FB (0==Local; 1==Remote)
        [2].13   // T2 Part Detect Indicator
        [2].9   // Accumulator Conveyor Status
        [70]   // Scaled Seam Position (0-100)
        [6].1   // Master Control Status Ind
        [159].0   // Active Recipe CL ON/OFF
        [43]   // Line-Start Total Boost Voltage (start boost - stop decay)
        [190]   // Active Recipe Conveyor Speed (ft/min x 10)
        [200]   // Closed-Loop FIFO Length FB
        [5].0   // Recipe Edit Handshake (To PV)
        [0].2   // Exit Exhaust VFD ON
        [112]   // IR Zone 3 Run Value
        [2].7   // Exhaust Air-Flow Switch
        [51]   // Oven Exit Pyrometer Temperature #1 Feedback (0-5Vdc == 32-932f)
        [55]   // Oven Exit Pyrometer Temperature #5 Feedback (0-5Vdc == 32-932f)
        [1].1   // Oven Conveyor Run Indicator
        [102]   // Oven Exhaust Speed Setpoint (0-100%)
        [2].2   // Oven Entrance Part Detect Indicator
        [50]   // Oven Temperature Feedback (0-10Vdc == 32-932f)
        [0].9   // Local/Remote Line Speed FB (0==Local)
        [151]   // Active Recipe Zone 2 Voltage
        [37]   // Duct Heater % Power Out (0 - 100)
        [152]   // Active Recipe Zone 3 Voltage
        [21]   // Control List Selector - Keep Equal to 0
        [113]   // IR Zone 4 Run Value
        [114]   // IR Zone 5 Run Value
        [115]   // IR Zone 6 Run Value
        [116]   // IR Zone 7 Run Value
        [117]   // IR Zone 8 Run Value
        [118]   // IR Zone 9 Run Value
        [156]   // Active Recipe Value 7
        [157]   // Active Recipe Value 8
        [158]   // Active Recipe Value 9
        [0].3   // Coooldown #1 Exhaust MS ON
        [215]   // VFD Exhst. TOTAL Correction (Hz)
        [101]   // Duct Heater Temperature Setpoint (32-932)
        [0].5   // Coooldown #2 Exhaust MS ON
        [1].2   // Cooldown Conveyor Run Indicator
        [192].0   // Active Recipe CL ON/OFF
        [214]   // VFD Exhst. Integral Correction (Hz)
        [153]   // Active Recipe Zone 4 Voltage
        [2].8   // Entrance Exit Air-Flow Switch
        [5].11   // Closed-Loop Control ON/OFF FB
        [195]   // Active Recipe Peak-Picker Delay
        [213]   // VFD Exhst. Proportional Correction (Hz)
        [103]   // Oven Recirculation Blower Speed Setpoint (0-100%)
        [52]   // Oven Exit Pyrometer Temperature #2 Feedback (0-5Vdc == 32-932f)
        [301]   // Closed-Loop Proportional Correction
        [191]   // Active Recipe Closed-Loop Temperature Setpoint
        [196]   // Active Recipe Peak-Picker Duration
        [198]   // Active Recipe Exhaust Duct Temperature Setpoint
        [2].6   // Cooldown Conveyor Motion Detect Indicator
        [154]   // Active Recipe Zone 5 Voltage
        [100]   // Oven Conveyor Run Value (0-600)
        [0].10   // System Ready Auto + Soak Timer DONE
   N28 : DINT[200] := ([10] := 6826, [11] := 6826, [12] := 6826, [13] := 6826, [14] := 6826, [15] := 6826, [16] := 6826, [17] := 6826, [50] := 100, [51] := 60, [52] := 350, [53] := 77, [60] := 150, [61] := 175, [62] := 175, [63] := 350, [64] := 350, [65] := 350);   // Read from PLC
        [100]   // Mapped Alarms to PV
        [2]   // Power Brush Speed Out (0-32767)
        [129]   // Closed-Loop #1 FIFO Value #10
        [139]   // Closed-Loop #2 FIFO Value #10
        [120]   // Closed-Loop #1 FIFO Value #1
        [10]   // Zone 1 Output (0-32767)
        [121]   // Closed-Loop #1 FIFO Value #2
        [122]   // Closed-Loop #1 FIFO Value #3
        [123]   // Closed-Loop #1 FIFO Value #4
        [124]   // Closed-Loop #1 FIFO Value #5
        [125]   // Closed-Loop #1 FIFO Value #6
        [126]   // Closed-Loop #1 FIFO Value #7
        [127]   // Closed-Loop #1 FIFO Value #8
        [128]   // Closed-Loop #1 FIFO Value #9
        [130]   // Closed-Loop #2 FIFO Value #1
        [131]   // Closed-Loop #2 FIFO Value #2
        [132]   // Closed-Loop #2 FIFO Value #3
        [19]   // Zone 10 Output (0-32767)
        [11]   // Zone 2 Output (0-32767)
        [12]   // Zone 3 Output (0-32767)
        [13]   // Zone 4 Output (0-32767)
        [14]   // Zone 5 Output (0-32767)
        [101]   // Mapped Alarms to PV
        [102]   // Mapped Alarms to PV
        [103]   // Mapped Alarms to PV
        [104]   // Mapped Alarms to PV
        [105]   // Mapped Alarms to PV
        [106]   // Mapped Alarms to PV
        [107]   // Mapped Alarms to PV
        [133]   // Closed-Loop #2 FIFO Value #4
        [0]   // Mapped Alarms to PV
        [134]   // Closed-Loop #2 FIFO Value #5
        [135]   // Closed-Loop #2 FIFO Value #6
        [136]   // Closed-Loop #2 FIFO Value #7
        [108]   // Mapped Alarms to PV
        [137]   // Closed-Loop #2 FIFO Value #8
        [15]   // Zone 6 Output (0-32767)
        [16]   // Zone 7 Output (0-32767)
        [17]   // Zone 8 Output (0-32767)
        [109]   // Mapped Alarms to PV
        [138]   // Closed-Loop #2 FIFO Value #9
        [1]   // Rotator Speed Out (0-32767)
        [18]   // Zone 9 Output (0-32767)
        [50]   // Recipe Edit Display
   N32 : DINT[200] := ([2] := 300, [3] := 51, [4] := 1, [5] := 50, [6] := 51, [9] := 20, [10] := 45, [20] := -75, [21] := 75, [24] := 1, [25] := 225, [40] := 7, [41] := 97, [42] := 54, [100] := 2147483647, [101] := 2147483623, [102] := 2147483647, [103] := 2147483647, [104] := 2147483647, [105] := 2147483647, [106] := 2147483647, [107] := 2147483647, [108] := 2147483647, [109] := 2147483647, [120] := 2147483647, [121] := 2147483623, [122] := 2147483647, [123] := 2147483647, [124] := 2147483647, [125] := 2147483647, [126] := 2147483647, [127] := 2147483647, [128] := 2147483647, [160] := 65535, [161] := 65535, [162] := 65535, [163] := 65535, [164] := 65535, [165] := 65535, [166] := 65535, [167] := 65535, [168] := 65535, [169] := 65535);
        [10]   // Recipe Edit Scaled Entry Value
        [12]   // Line-Start Boost Voltage to ADD
        [9]   // Previous Recipe to Be Edited
        [5]   // Address Offset Compute
        [20]   // Closed-Loop #1 Max. Negative Boost Voltage
        [25]   // 1st Closed-Loop FIFO Average
        [11]   // Line-Start Boost % Power to ADD
        [4]   // File Offset Compute
        [35]   // 2nd Closed-Loop FIFO Average
        [24]   // Closed-Loop #1 FIFO Loop Adder
        [13]   // Line-Stop Boost % Power to SUBTRACT
        [3]   // Integer File Offset (All Recipe Storage begins @ N50:00)
        [34]   // Closed-Loop #2 FIFO Loop Adder
        [23]   // Closed-Loop #1 Pyrometer Peak-Picker
        [1]   // Recipe to Run Offset Value
        [33]   // Closed-Loop #2 Pyrometer Peak-Picker
        [22]   // Peak Temperature
        [14]   // Line-Stop Boost Voltage SUBTRACT
        [2]   // Get Recipe Indexed Offset
        [21]   // Closed-Loop #1 Max. Positive Boost Voltage
        [0]   // Recipe Offset
        [42]   // Actuator Movement in the last 4 seconds
        [26]   // Closed-Loop #1 FIFO Temperature Difference
        [30]   // Closed-Loop #2 Max. Negative Boost Voltage
        [41]   // Seam Actuator Movement Check Value
        [31]   // Closed-Loop #2 Max. Positive Boost Voltage
        [100]   // Alarm Horn Mask Compare Value
        [130]   // Alarm Horn Compare Result
        [6]   // File Offset
        [36]   // Closed-Loop #2 FIFO Temperature Difference
        [27]   // FIFO Ave Intermediary Register
   N32_1 : DINT;   // Recipe to Run Offset Value
   N32_2 : DINT;   // Recipe Copy Utility
   N32_3 : DINT := 450;   // Recipe Copy Utility
   N40 : DINT[256] := ([0] := 20, [1] := 20, [2] := 20, [3] := 20, [4] := 20, [5] := 20, [6] := 20, [7] := 20, [8] := 20, [9] := 20, [10] := 20, [11] := 20, [12] := 20, [13] := 20, [14] := 20, [15] := 20, [16] := 20, [17] := 20, [18] := 20, [19] := 20, [20] := 20, [21] := 20, [22] := 20, [23] := 20, [24] := 20, [25] := 20, [26] := 20, [27] := 20, [28] := 20, [29] := 20, [30] := 20, [31] := 20, [32] := 20, [33] := 20, [34] := 20, [35] := 20, [36] := 20, [37] := 20, [38] := 20, [39] := 20, [40] := 20, [41] := 20, [42] := 20, [43] := 20, [44] := 20, [45] := 20, [46] := 20, [47] := 20, [48] := 20, [49] := 20, [50] := 20, [51] := 20, [52] := 20, [53] := 20, [54] := 20, [55] := 20, [56] := 20, [57] := 20, [58] := 20, [59] := 20,
        [60] := 20, [61] := 20, [62] := 20, [63] := 20, [64] := 20, [65] := 20, [66] := 20, [67] := 20, [68] := 20, [69] := 20, [70] := 20, [71] := 20, [72] := 20, [73] := 20, [74] := 20, [75] := 20, [76] := 20, [77] := 20, [78] := 20, [79] := 20, [80] := 20, [81] := 20, [82] := 20, [83] := 20, [84] := 20, [85] := 20, [86] := 20, [87] := 20, [88] := 20, [89] := 20, [90] := 20, [91] := 20, [92] := 20, [93] := 20, [94] := 20, [95] := 20, [96] := 20, [97] := 20, [98] := 20, [99] := 20, [100] := 20, [101] := 20, [102] := 20, [103] := 20, [104] := 20, [105] := 20, [106] := 20, [107] := 20, [108] := 20, [109] := 20, [110] := 20, [111] := 20, [112] := 20, [113] := 20, [114] := 20, [115] := 20, [116] := 20, [117] := 20, [118] := 20, [119] := 20,
        [120] := 20, [121] := 20, [122] := 20, [123] := 20, [124] := 20, [125] := 20, [126] := 20, [127] := 20, [128] := 20, [129] := 20, [130] := 20, [131] := 20, [132] := 20, [133] := 20, [134] := 20, [135] := 20, [136] := 20, [137] := 20, [138] := 20, [139] := 20, [140] := 20, [141] := 20, [142] := 20, [143] := 20, [144] := 20, [145] := 20, [146] := 20, [147] := 20, [148] := 20, [149] := 20, [150] := 20, [151] := 20, [152] := 20, [153] := 20, [154] := 20, [155] := 20, [156] := 20, [157] := 20, [158] := 20, [159] := 20, [160] := 20, [161] := 20, [162] := 20, [163] := 20, [164] := 20, [165] := 20, [166] := 20, [167] := 20, [168] := 20, [169] := 20, [170] := 20, [171] := 20, [172] := 20, [173] := 20, [174] := 20, [175] := 20, [176] := 20, [177] := 20, [178] := 20, [179] := 20,
        [180] := 20, [181] := 20, [182] := 20, [183] := 20, [184] := 20, [185] := 20, [186] := 20, [187] := 20, [188] := 20, [189] := 20, [190] := 20, [191] := 20, [192] := 20, [193] := 20, [194] := 20, [195] := 20, [196] := 20, [197] := 20, [198] := 20, [199] := 20, [200] := 20, [201] := 20, [202] := 20, [203] := 20, [204] := 20, [205] := 20, [206] := 20, [207] := 20, [208] := 20, [209] := 20, [210] := 20, [211] := 20, [212] := 20, [213] := 20, [214] := 20, [215] := 20, [216] := 20, [217] := 20, [218] := 20, [219] := 20, [220] := 20, [221] := 20, [222] := 20, [223] := 20, [224] := 20, [225] := 20, [226] := 20, [227] := 20, [228] := 20, [229] := 20, [230] := 20, [231] := 20, [232] := 20, [233] := 20, [234] := 20, [235] := 20, [236] := 20, [237] := 20, [238] := 20, [239] := 20,
        [240] := 20, [241] := 20, [242] := 20, [243] := 20, [244] := 20, [245] := 20, [246] := 20, [247] := 20, [248] := 20, [249] := 20, [250] := 20, [251] := 20, [252] := 20, [253] := 20, [254] := 20);   // Recipe Shift
        [129]   // Recipe Shift
        [0]   // Recipe Shift
        [1]   // Recipe Shift
   N41 : DINT[256] := ([0] := 20, [1] := 20, [2] := 20, [3] := 20, [4] := 20, [5] := 20, [6] := 20, [7] := 20, [8] := 20, [9] := 20, [10] := 20, [11] := 20, [12] := 20, [13] := 20, [14] := 20, [15] := 20, [16] := 20, [17] := 20, [18] := 20, [19] := 20, [20] := 20, [21] := 20, [22] := 20, [23] := 20, [24] := 20, [25] := 20, [26] := 20, [27] := 20, [28] := 20, [29] := 20, [30] := 20, [31] := 20, [32] := 20, [33] := 20, [34] := 20, [35] := 20, [36] := 20, [37] := 20, [38] := 20, [39] := 20, [40] := 20, [41] := 20, [42] := 20, [43] := 20, [44] := 20, [45] := 20, [46] := 20, [47] := 20, [48] := 20, [49] := 20, [50] := 20, [51] := 20, [52] := 20, [53] := 20, [54] := 20, [55] := 20, [56] := 20, [57] := 20, [58] := 20, [59] := 20,
        [60] := 20, [61] := 20, [62] := 20, [63] := 20, [64] := 20, [65] := 20, [66] := 20, [67] := 20, [68] := 20, [69] := 20, [70] := 20, [71] := 20, [72] := 20, [73] := 20, [74] := 20, [75] := 20, [76] := 20, [77] := 20, [78] := 20, [79] := 20, [80] := 20, [81] := 20, [82] := 20, [83] := 20, [84] := 20, [85] := 20, [86] := 20, [87] := 20, [88] := 20, [89] := 20, [90] := 20, [91] := 20, [92] := 20, [93] := 20, [94] := 20, [95] := 20, [96] := 20, [97] := 20, [98] := 20, [99] := 20, [100] := 20, [101] := 20, [102] := 20, [103] := 20, [104] := 20, [105] := 20, [106] := 20, [107] := 20, [108] := 20, [109] := 20, [110] := 20, [111] := 20, [112] := 20, [113] := 20, [114] := 20, [115] := 20, [116] := 20, [117] := 20, [118] := 20, [119] := 20,
        [120] := 20, [121] := 20, [122] := 20, [123] := 20, [124] := 20, [125] := 20, [126] := 20, [127] := 20, [128] := 20, [129] := 20, [130] := 20, [131] := 20, [132] := 20, [133] := 20, [134] := 20, [135] := 20, [136] := 20, [137] := 20, [138] := 20, [139] := 20, [140] := 20, [141] := 20, [142] := 20, [143] := 20, [144] := 20, [145] := 20, [146] := 20, [147] := 20, [148] := 20, [149] := 20, [150] := 20, [151] := 20, [152] := 20, [153] := 20, [154] := 20, [155] := 20, [156] := 20, [157] := 20, [158] := 20, [159] := 20, [160] := 20, [161] := 20, [162] := 20, [163] := 20, [164] := 20, [165] := 20, [166] := 20, [167] := 20, [168] := 20, [169] := 20, [170] := 20, [171] := 20, [172] := 20, [173] := 20, [174] := 20, [175] := 20, [176] := 20, [177] := 20, [178] := 20, [179] := 20,
        [180] := 20, [181] := 20, [182] := 20, [183] := 20, [184] := 20, [185] := 20, [186] := 20, [187] := 20, [188] := 20, [189] := 20, [190] := 20, [191] := 20, [192] := 20, [193] := 20, [194] := 20, [195] := 20, [196] := 20, [197] := 20, [198] := 20, [199] := 20, [200] := 20, [201] := 20, [202] := 20, [203] := 20, [204] := 20, [205] := 20, [206] := 20, [207] := 20, [208] := 20, [209] := 20, [210] := 20, [211] := 20, [212] := 20, [213] := 20, [214] := 20, [215] := 20, [216] := 20, [217] := 20, [218] := 20, [219] := 20, [220] := 20, [221] := 20, [222] := 20, [223] := 20, [224] := 20, [225] := 20, [226] := 20, [227] := 20, [228] := 20, [229] := 20, [230] := 20, [231] := 20, [232] := 20, [233] := 20, [234] := 20, [235] := 20, [236] := 20, [237] := 20, [238] := 20, [239] := 20,
        [240] := 20, [241] := 20, [242] := 20, [243] := 20, [244] := 20, [245] := 20, [246] := 20, [247] := 20, [248] := 20, [249] := 20);   // Recipe Shift
        [126]   // Recipe Shift
        [0]   // Recipe Shift
        [1]   // Recipe Shift
   N42 : DINT[256] := ([0] := 20, [1] := 20, [2] := 20, [3] := 20, [4] := 20, [5] := 20, [6] := 20, [7] := 20, [8] := 20, [9] := 20, [10] := 20, [11] := 20, [12] := 20, [13] := 20, [14] := 20, [15] := 20, [16] := 20, [17] := 20, [18] := 20, [19] := 20, [20] := 20, [21] := 20, [22] := 20, [23] := 20, [24] := 20, [25] := 20, [26] := 20, [27] := 20, [28] := 20, [29] := 20, [30] := 20, [31] := 20, [32] := 20, [33] := 20, [34] := 20, [35] := 20, [36] := 20, [37] := 20, [38] := 20, [39] := 20, [40] := 20, [41] := 20, [42] := 20, [43] := 20, [44] := 20, [45] := 20, [46] := 20, [47] := 20, [48] := 20, [49] := 20, [50] := 20, [51] := 20, [52] := 20, [53] := 20, [54] := 20, [55] := 20, [56] := 20, [57] := 20, [58] := 20, [59] := 20,
        [60] := 20, [61] := 20, [62] := 20, [63] := 20, [64] := 20, [65] := 20, [66] := 20, [67] := 20, [68] := 20, [69] := 20, [70] := 20, [71] := 20, [72] := 20, [73] := 20, [74] := 20, [75] := 20, [76] := 20, [77] := 20, [78] := 20, [79] := 20, [80] := 20, [81] := 20, [82] := 20, [83] := 20, [84] := 20, [85] := 20, [86] := 20, [87] := 20, [88] := 20, [89] := 20, [90] := 20, [91] := 20, [92] := 20, [93] := 20, [94] := 20, [95] := 20, [96] := 20, [97] := 20, [98] := 20, [99] := 20, [100] := 20, [101] := 20, [102] := 20, [103] := 20, [104] := 20, [105] := 20, [106] := 20, [107] := 20, [108] := 20, [109] := 20, [110] := 20, [111] := 20, [112] := 20, [113] := 20, [114] := 20, [115] := 20, [116] := 20, [117] := 20, [118] := 20, [119] := 20,
        [120] := 20, [121] := 20, [122] := 20, [123] := 20, [124] := 20, [125] := 20, [126] := 20, [127] := 20, [128] := 20, [129] := 20, [130] := 20, [131] := 20, [132] := 20, [133] := 20, [134] := 20, [135] := 20, [136] := 20, [137] := 20, [138] := 20, [139] := 20, [140] := 20, [141] := 20, [142] := 20, [143] := 20, [144] := 20, [145] := 20, [146] := 20, [147] := 20, [148] := 20, [149] := 20, [150] := 20, [151] := 20, [152] := 20, [153] := 20, [154] := 20, [155] := 20, [156] := 20, [157] := 20, [158] := 20, [159] := 20, [160] := 20, [161] := 20, [162] := 20, [163] := 20, [164] := 20, [165] := 20, [166] := 20, [167] := 20, [168] := 20, [169] := 20, [170] := 20, [171] := 20, [172] := 20, [173] := 20, [174] := 20, [175] := 20, [176] := 20, [177] := 20, [178] := 20, [179] := 20,
        [180] := 20, [181] := 20, [182] := 20, [183] := 20, [184] := 20, [185] := 20, [186] := 20, [187] := 20, [188] := 20, [189] := 20, [190] := 20, [191] := 20, [192] := 20, [193] := 20, [194] := 20, [195] := 20, [196] := 20, [197] := 20, [198] := 20, [199] := 20, [200] := 20, [201] := 20, [202] := 20, [203] := 20, [204] := 20, [205] := 20, [206] := 20, [207] := 20, [208] := 20, [209] := 20, [210] := 20, [211] := 20, [212] := 20, [213] := 20, [214] := 20, [215] := 20, [216] := 20, [217] := 20, [218] := 20, [219] := 20, [220] := 20, [221] := 20, [222] := 20, [223] := 20, [224] := 20, [225] := 20, [226] := 20, [227] := 20, [228] := 20, [229] := 20, [230] := 20, [231] := 20, [232] := 20, [233] := 20, [234] := 20, [235] := 20, [236] := 20, [237] := 20, [238] := 20, [239] := 20,
        [240] := 20, [241] := 20, [242] := 20, [243] := 20, [244] := 20, [245] := 20, [246] := 20, [247] := 20, [248] := 20, [249] := 20, [250] := 20, [251] := 20, [252] := 20, [253] := 20, [254] := 20);   // Recipe Shift
        [125]   // Recipe Shift
        [128]   // Recipe Shift
        [0]   // Recipe Shift
   N50 : DINT[2500] := ([0] := 400, [1] := 400, [2] := 400, [3] := 400, [4] := 400, [5] := 400, [6] := 400, [7] := 360, [8] := 360, [40] := 40, [41] := 400, [42] := 40, [43] := 100, [45] := 30, [46] := 8, [47] := 1, [48] := 275, [50] := 400, [51] := 400, [52] := 400, [53] := 400, [54] := 400, [55] := 400, [56] := 400, [57] := 360, [58] := 360, [90] := 59, [91] := 351, [92] := 49, [93] := 50, [95] := 30, [96] := 8, [97] := 1, [98] := 275, [100] := 400, [101] := 400, [102] := 400, [103] := 400, [104] := 400, [105] := 400, [106] := 400, [107] := 360, [108] := 360, [140] := 15, [141] := 230, [142] := 20, [143] := 25, [145] := 30, [146] := 8, [147] := 1, [148] := 275, [150] := 400, [151] := 400, [152] := 400, [153] := 400, [154] := 400, [155] := 400, [156] := 400, [157] := 360, [158] := 360,
        [190] := 15, [191] := 230, [192] := 20, [193] := 25, [195] := 30, [196] := 8, [197] := 1, [198] := 275, [200] := 400, [201] := 400, [202] := 400, [203] := 400, [204] := 400, [205] := 400, [206] := 400, [207] := 360, [208] := 360, [240] := 15, [241] := 230, [242] := 20, [243] := 25, [245] := 30, [246] := 8, [247] := 1, [248] := 275, [250] := 400, [251] := 400, [252] := 400, [253] := 400, [254] := 400, [255] := 400, [256] := 400, [257] := 360, [258] := 360, [290] := 15, [291] := 230, [292] := 20, [293] := 25, [295] := 30, [296] := 8, [297] := 1, [298] := 275, [300] := 400, [301] := 400, [302] := 400, [303] := 400, [304] := 400, [305] := 400, [306] := 400, [307] := 360, [308] := 360, [340] := 15, [341] := 230, [342] := 20, [343] := 25, [345] := 30, [346] := 8, [347] := 1, [348] := 275, [350] := 400,
        [351] := 400, [352] := 400, [353] := 400, [354] := 400, [355] := 400, [356] := 400, [357] := 360, [358] := 360, [390] := 15, [391] := 230, [392] := 20, [393] := 25, [395] := 30, [396] := 8, [397] := 1, [398] := 275, [400] := 400, [401] := 400, [402] := 400, [403] := 400, [404] := 400, [405] := 400, [406] := 400, [407] := 360, [408] := 360, [440] := 15, [441] := 230, [442] := 20, [443] := 25, [445] := 30, [446] := 8, [447] := 1, [448] := 275, [450] := 400, [451] := 400, [452] := 400, [453] := 400, [454] := 400, [455] := 400, [456] := 400, [457] := 360, [458] := 360, [490] := 15, [491] := 230, [492] := 20, [493] := 25, [495] := 30, [496] := 8, [497] := 1, [498] := 275, [500] := 450, [501] := 450, [502] := 450, [503] := 450, [504] := 450, [505] := 450, [506] := 450, [507] := 450, [508] := 450, [540] := 25,
        [541] := 230, [542] := 1, [545] := 10, [546] := 15, [547] := 1, [548] := 275, [550] := 230, [551] := 230, [552] := 230, [553] := 230, [554] := 230, [555] := 230, [556] := 230, [557] := 230, [558] := 230, [590] := 20, [591] := 230, [592] := 1, [595] := 3, [596] := 12, [597] := 1, [598] := 230, [600] := 1, [601] := 1, [602] := 1, [603] := 1, [604] := 1, [605] := 1, [606] := 1, [607] := 1, [608] := 1, [640] := 15, [641] := 215, [645] := 7, [646] := 12, [647] := 1, [648] := 340, [690] := 16, [691] := 16, [692] := 1, [695] := 3, [696] := 5, [700] := 450, [701] := 450, [702] := 450, [703] := 450, [704] := 450, [705] := 450, [706] := 450, [707] := 450, [708] := 450, [710] := 100, [711] := 100, [712] := 100, [713] := 400, [714] := 400, [715] := 400, [740] := 25, [741] := 250, [742] := 1,
        [745] := 25, [746] := 15, [747] := 1, [748] := 275, [750] := 340, [751] := 340, [753] := 340, [754] := 340, [760] := 100, [761] := 100, [762] := 100, [763] := 400, [764] := 400, [765] := 400, [790] := 25, [791] := 215, [792] := 1, [795] := 3, [796] := 8, [800] := 315, [801] := 315, [802] := 315, [803] := 315, [804] := 315, [805] := 315, [840] := 34, [841] := 205, [842] := 1, [845] := 5, [846] := 10, [850] := 400, [851] := 375, [853] := 400, [854] := 375, [890] := 27, [891] := 215, [892] := 1, [895] := 10, [896] := 12, [900] := 390, [901] := 390, [903] := 390, [904] := 390, [940] := 28, [941] := 215, [942] := 1, [945] := 8, [946] := 8, [950] := 330, [951] := 330, [953] := 330, [954] := 330, [990] := 40, [991] := 120, [992] := 45, [993] := 75, [995] := 5, [996] := 8, [1000] := 280, [1001] := 280,
        [1003] := 380, [1004] := 380, [1040] := 28, [1041] := 215, [1042] := 1, [1045] := 3, [1046] := 5, [1050] := 350, [1051] := 350, [1053] := 350, [1054] := 350, [1090] := 35, [1091] := 215, [1092] := 1, [1095] := 5, [1096] := 8, [1200] := 330, [1201] := 330, [1203] := 330, [1204] := 330, [1240] := 28, [1241] := 215, [1242] := 1, [1245] := 5, [1246] := 8, [1450] := 30, [1455] := 30, [1490] := 30, [1950] := 250, [1951] := 175, [1952] := 125, [1953] := 250, [1954] := 75, [1955] := 75, [1956] := 250, [1957] := 75, [1958] := 75, [1990] := 10, [1991] := 150, [1998] := 150, [2390] := 10, [2400] := 50, [2401] := 50, [2402] := 50, [2403] := 50, [2404] := 50, [2405] := 50, [2406] := 50, [2407] := 50, [2408] := 50, [2440] := 20, [2441] := 32, [2445] := 15, [2446] := 15, [2447] := 1, [2448] := 150, [2450] := 50, [2451] := 50, [2452] := 50, [2453] := 50,
        [2454] := 50, [2455] := 50, [2456] := 50, [2457] := 50, [2458] := 50, [2490] := 150, [2491] := 235, [2492] := 1, [2495] := 25, [2496] := 10, [2497] := 1, [2498] := 225);   // Stored Recipes
        [0]   // Stored Recipes
   N7 : DINT[250] := ([10] := 111, [20] := 1819, [21] := 1819, [22] := 53, [24] := 8160, [26] := 235, [30] := 4000, [31] := -8, [32] := 3000, [35] := 390, [36] := 410, [37] := 400, [38] := 75, [41] := 8, [42] := 75, [50] := 300);   // Utility Integers
        [0]   // Zone1 Power (0-31206)
        [1]   // Zone2 Power (0-31206)
        [10]   // T2 Zone11 Power (0-32767)
        [9]   // T1 Zone10 Power (0-32767)
        [12]   // T2 Zone1 Power (0-32767)
        [5]   // Zone 6 Power (0-31206)
        [8]   // Zone 9 Power (0-32767)
        [30]   // FIFO Reset Distance
        [13]   // T1 Zone2 Power (0-32767)
        [14]   // T1 Zone3 Power (0-32767)
        [15]   // T1 Zone4 Power (0-32767)
        [16]   // T1 Zone5 Power (0-32767)
        [25]   // Temporary Math Register for CL Correction
        [37]   // Previous Temperature Setpoint
        [35]   // Temperature Soak Lower Limit
        [31]   // Oven Exhaust Temperature Above Setpoint
        [27]   // Purge Time Remaining
        [33]   // Duct Heater Output
        [11]   // T1 Zone12 Power (0-32767)
        [36]   // Temperature Soak Upper Limit
        [24]   // Exhaust Temperature Raw Data Feedback
        [40]   // T1 Conveyor Speed (0-32767)
        [21]   // Oven Exit Part Raw Temperature Feedback - 6234
        [17]   // T1 Zone6 Power (0-32767)
        [32]   // Integral Corr'n Time - 0.001s
        [20]   // Oven Exit Part Raw Temperature Feedback
        [2]   // Zone3 Power (0-31206)
        [22]   // Raw Feedback (N7[21]) * Scaling
        [3]   // Zone4 Power (0-31206)
        [4]   // Zone5 Power (0-31206)
        [6]   // Zone7 Power (0-32767)
        [7]   // Zone8 Power (0-32767)
        [38]   // Previous VFD Setpoint
        [26]   // Raw Feedback (N7[24]) * Scaling
        [41]   // Oven Exhaust Temperature Below Setpoint
        [42]   // VFD Auto Mode Corrected Output (0-100%)
        [50]   // Cooldown Blowers Start Distance from IR Section 3 Start
   o2 : INT[8] := ([4] := 12757);   // Slot 2 8-pt Analog Output
        [2]   // Spare (0-10Vdc)
        [0]   // Oven Conveyor Speed (0-10Vdc)
        [6]   // Spare (0-10Vdc)
        [7]   // Spare (0-10Vdc)
        [4]   // Duct Heater Remote Setpoint (0-10Vdc == 32-932f)
        [1]   // Exhaust VFD Speed (0-10Vdc)
        [3]   // Recirculation Blower VFD Speed (0-10Vdc)
        [5]   // BGK Conveyor Speed Reference to Customer (0-10Vdc)
   o5 : SINT := 48;   // Slot 5 8-pt Relay Output
        .4   // UV Trip Enable
        .1   // Light Stack Red - System Fault
        .2   // Light Stack Amber - System In Manual
        .6   // Spare
        .5   // MCR Enable
        .0   // Fault Horn
        .3   // Light Stack Green - System Running
        .7   // Spare
   o6 : SINT;   // Slot 6 8-pt Relay Output
        .4   // Spare
        .1   // HEPA Supply Blowers RUN
        .5   // Recirculation VFD Run
        .3   // Exhaust VFD Run Enable
        .2   // Oven Conveyor VFD RUN
        .7   // Spare
        .0   // Duct Heater Enable
        .6   // BGK Oven Ready to Customer
   Offset : DINT := 950;
   Oven_Exhaust_Temp_Raw : INT := 8160;   // Move the last 16 bits of Double Integer i1[0]
   Oven_Exhaust_Temp_Scaled : INT;
   Oven_Exit_Temp_Raw : INT := 1819;   // Move the 1st 16 bits of Double Integer i1[0]
   Oven_Exit_Temp_Scaled : INT;
   R6 : CONTROL[10] := ([0].LEN := 128, [0].POS := 127, [1].LEN := 2048, [2].LEN := 7);
        [1]   // B10 is the part Location Shift File
   S24 : INT := 16#0003;   // Index Register
   T24 : TIMER[150] := ([5].PRE := 75000, [6].PRE := 750, [7].PRE := 3000, [8].PRE := 3000, [10].PRE := 500, [11].PRE := 15000, [12].PRE := 55000, [13].PRE := 500, [14].PRE := 15000, [15].PRE := 55000, [16].PRE := 5000, [17].PRE := 5000, [18].PRE := 5000, [19].PRE := 5000, [20].PRE := 5000, [21].PRE := 5000, [22].PRE := 5000, [23].PRE := 5000, [24].PRE := 5000, [25].PRE := 5000, [26].PRE := 1500, [27].PRE := 350, [28].PRE := 15000, [39].PRE := 2000, [40].PRE := 2000, [41].PRE := 500000, [42].PRE := 500000, [49].PRE := 100, [50].PRE := 100, [51].PRE := 100, [52].PRE := 100, [53].PRE := 100, [54].PRE := 20, [55].PRE := 10, [56].PRE := 20, [58].PRE := 20, [59].PRE := 20, [60].PRE := 2000, [61].PRE := 5000, [62].PRE := 5000, [62].ACC := 64, [62].EN := 1, [62].TT := 1, [63].PRE := 10, [70].PRE := 50, [71].PRE := 50, [72].PRE := 50, [73].PRE := 50, [73].ACC := 50, [74].PRE := 50, [75].PRE := 50, [76].PRE := 50, [77].PRE := 50, [78].PRE := 50, [79].PRE := 100, [80].PRE := 500, [80].ACC := 500, [80].EN := 1, [80].DN := 1, [83].PRE := 200,
        [83].ACC := 201, [83].EN := 1, [83].DN := 1, [84].PRE := 200, [84].ACC := 201, [84].EN := 1, [84].DN := 1, [85].PRE := 200, [85].ACC := 201, [85].EN := 1, [85].DN := 1, [90].PRE := 500, [91].PRE := 350, [92].PRE := 350, [92].ACC := 351, [92].EN := 1, [92].DN := 1, [93].PRE := 350, [94].PRE := 250, [95].PRE := 3000, [96].PRE := 8000);   // Fault Timers
        [50]   // Cooldown Conveyor VFD Disconnect Fault
        [5]   // Temperature Deviation Fault
        [25]   // P5 High Temp Warning
        [41]   // ENTRANCE PART STOPPED FAULT
        [70]   // Booth #1 Fire Detect
        [49]   // IR Conveyor VFD Disconnect Fault
        [42]   // EXIT PART STOPPED FAULT
        [95]   // MCR NOT ON FAULT DELAY
        [24]   // P4 High Temp Warning
        [23]   // P3 High Temp Warning
        [14]   // IR Exhaust Air-Flow Fault
        [15]   // IR Exhaust Air-Flow Switch Fault
        [54]   // Conveyor Jam/Take-Up Fault
        [58]   // Spindle NOT Seated at Loader Fualt
        [79]   // Oven Doors Open Fault
        [78]   // Spray Booth Line-Stop Fault
        [55]   // Part On Spindle Before Loader Fault
        [92]   // Remote Console E-Stop
        [76]   // Loader Line-Stop Fault
        [93]   // Oven Lift Disconnect Fault
        [17]   // P2 Low Temp Warning
        [72]   // Booth #1 Low Powder
        [74]   // Booth #2 Not Ready
        [21]   // P1 High Temp Warning
        [52]   // PEG Conveyor VFD Disconnect Fault
        [39]   // Oven Conveyor VFD Faulted
        [73]   // Booth #2 Fire Detect
        [26]   // T2 IR Supply #2 MS Fault
        [75]   // Booth #2 Low Powder
        [40]   // Cooldown Conveyor VFD Faulted
        [60]   // IR Conveyor Motion Fault
        [80]   // E-Stop Pressed Fault
        [62]   // Cooldown Conveyor Motion Fault
        [59]   // Filter Jammed at Loader Screw Fault
        [61]   // IR Conveyor Motion Fault
        [10]   // Recirculation VFD Fault
        [71]   // Spray Booth #1 Not Ready
        [11]   // Recirculation Air-Flow Fault
        [83]   // T2 Conveyor Load Line-Stop
        [91]   // Main CB UV Enable
        [84]   // T2 Conveyor UnLoad Line-Stop
        [63]   // Seam Heater Crash Detect Fault
        [94]   // Oven Lift Open Fault Timer
        [13]   // IR Exhaust VFD MS Fault
        [53]   // T2 Exhaust VFD Disconnect Fault
        [27]   // Main CB UV Enable
        [100]   // Seam Movement Check Timer
        [20]   // P5 Low Temp Warning
        [16]   // P1 Low Temp Warning
        [19]   // P4 Low Temp Warning
        [18]   // P3 Low Temp Warning
        [104]   // Control Panel Door E-Stop Fault
        [22]   // P2 High Temp Warning
        [12]   // Recirculation Air-Flow Switch Fault
        [28]   // T2 IR Supply #2 Air-Flow Switch Fault
        [77]   // Unloader Line-Stop Fault
        [51]   // Exhaust VFD Disconnect Fault
        [85]   // Line Stop Washer Conveyor Load End Fault
        [96]   // OVEN CONVEYOR NOT ON DELAY
        [90]   // MAIN CAB DISC OFF OR HIGH TEMP LIMIT IS TRIPPED DELAY
        [6]   // Oven Overtemp Limit Fault
        [7]   // Hot-Air Contactor #1 Fault
        [8]   // Hot-Air Contactor #2 Fault
   T34 : TIMER[30] := ([0].PRE := 1000, [0].ACC := 1000, [0].EN := 1, [0].DN := 1, [1].PRE := 250, [1].ACC := 251, [1].EN := 1, [1].DN := 1, [2].PRE := 250, [3].PRE := 250, [4].PRE := 1000, [4].ACC := 1000, [4].EN := 1, [4].DN := 1, [5].PRE := 1500, [6].PRE := 1500, [7].PRE := 1500, [8].PRE := 125, [9].PRE := 15000, [10].PRE := 250, [10].EN := 1, [10].DN := 1, [11].PRE := 15000, [14].PRE := 250, [15].PRE := 60000, [16].PRE := 100, [17].PRE := 1000, [18].PRE := 100, [18].ACC := 100, [20].PRE := 3000, [21].PRE := 500, [22].PRE := 500, [23].PRE := 3000, [24].PRE := 3000, [24].ACC := 3001, [24].EN := 1, [24].DN := 1, [26].PRE := 32767000, [26].ACC := 13573595, [26].EN := 1, [26].TT := 1, [27].PRE := 32767000, [27].ACC := 13847036, [27].EN := 1, [27].TT := 1);   // Utility Timers
        [4]   // Product Detect Timer
        [2].DN   // Product Detect Timer
        [11]   // Oven Purge Timer
        [1]   // MCR-On Timer
        [16]   // CLDN #2 Start Delay
        [12]   // C.L. #2 Conveyor Stop-Time Timer
        [18]   // CLDN #4 Start Delay
        [10]   // IR Oven Cooldown Timer
        [0]   // Power-On Timer
        [20].DN   // Conveyor Pre-Motion Timer
        [21].TT   // Pre-Motion Cascade Timer #1
        [8]   // Pseudo Motion Timer #2
        [17]   // T2 MCR-On Timer
        [27]   // Line-Stop Boost Timer
        [3]   // IR Recirculation Start Delay
        [26]   // Line-Start Boost Timer
        [23].DN   // Conveyor Startup Motion Fault Delay Done
        [5]   // Exhaust Start Delay
        [7]   // HEPA Supply Blowers Start Delay
        [14]   // Exit Product Detect Timer
        [6]   // Exit Exhaust Start Delay
        [23]   // Conveyor Startup Motion Fault Delay
        [21].EN   // Pre-Motion Cascade Timer #1
        [10].TT   // IR Oven Cooldown Timer
        [20]   // Conveyor Pre-Motion Timer
        [21]   // Pre-Motion Cascade Timer #1
        [22]   // Pre-Motion Cascade Timer #2
        [15]   // Horn on too long
        [9]   // C.L. #1 Conveyor Stop-Time Timer
        [24]   // Cooldown Conveyor Startup Motion Fault Delay
        [2]   // Entrance Product Detect Timer
   T4 : TIMER[32] := ([0].PRE := 60, [1].PRE := 500, [2].PRE := 14000, [3].PRE := 8000, [4].PRE := 8000, [6].PRE := 250, [7].PRE := 250, [8].PRE := 3000, [8].ACC := 2286, [8].EN := 1, [8].TT := 1, [10].PRE := 1500, [11].PRE := 15000, [20].PRE := 2100000000, [20].ACC := 28938197, [21].PRE := 2100000000, [21].ACC := 1033635448, [21].EN := 1, [21].TT := 1, [31].PRE := 10);
        [4]   // MinuteTimer Reset PB
        [3]   // Hour Timer Reset PB
        [1]   // Motion Simulate Timer
        [0].DN   // Feed Start Delay Time Done
        [0]   // Spare
        [31]   // SCR Fault Delay Timer
        [2]   // 14s Audible Cycle Timer
        [2].DN   // Meter Feed Start Delay Time Done
        [3].DN   // Meter Feed Stop Delay Time Done
        [10]   // Conveyor Start Bit Clear Timer
        [16]   // Pre-Cycle Timer #2
        [20]   // Oven ON Test Timer
        [5]   // Spare
        [8]   // VFD Integral Correction Timer
        [31].DN   // SCR Fault Delay Timer Done
        [24]   // Spare
        [15]   // Pre-Cycle Timer #1
        [21]   // Oven OFF Test Timer
        [12]   // Spare
        [25]   // Spare
        [13]   // Spare
        [14]   // Spare
        [9]   // Spare
        [26]   // Spare
        [6]   // Oven Exit Part Detect Nuisance Timer
        [7]   // FIFO Reset Part Detect Nuisance Timer
        [27]   // Spare
        [28]   // Spare
        [29]   // Spare
        [17]   // Spare
        [18]   // Spare
        [19]   // Spare
        [30]   // Spare
        [22]   // Spare
        [23]   // Spare
        [11]   // Hot-Air Soak Timer
   Test_Real : REAL := 288.40607;   // Temperature range (900/raw Data 4-20ma & 0-10v Range ma=(6241-31206) V= (0-31206)
END_VAR
